KUKA KRL program: nplacestr5RS2.src, nplacestr5RS2.dat

--- nplacestr5RS2.src ---
&ACCESS RVP
&REL 1
&PARAM TEMPLATE = C:\KRC\Roboter\Template\ExpertVorgabe
&PARAM EDITMASK = *
DEF nplacestr5RS2( )
;FOLD INI
  ;FOLD BASISTECH INI
    GLOBAL INTERRUPT DECL 3 WHEN $STOPMESS==TRUE DO IR_STOPM ( )
    INTERRUPT ON 3
    BAS (#INITMOV,0 )
  ;ENDFOLD (BASISTECH INI)
  ;FOLD USER INI
    ;Make your modifications here

  ;ENDFOLD (USER INI)
;ENDFOLD (INI)




SWITCH NumCuring

;*******************************************************
CASE 90501
;*******************************************************
;*** Utilizar para hacer touchup en ptp a continuacion ***;
; 1  Ejecutar Axis_Rob_Move
; 2  Hacer TouchUp en ptp
; 3  Eliminar Axis_Rob_Move y comentarios

Axis_Rob_Move(1.69,-82.8,66.93,14.32,12.14,193,70,50)

;FOLD PTP pWB90501RS2 Vel=100 % PDAT_MESA Tool[10]:AMF1_G1000 Base[9]:BWB2S2;%{PE}%R 5.5.32,%MKUKATPBASIS,%CMOVE,%VPTP,%P 1:PTP, 2:pWB90501RS2, 3:, 5:100, 7:PDAT_MESA
$BWDSTART=FALSE
PDAT_ACT=PPDAT_MESA
FDAT_ACT=FpWB90501RS2
BAS(#PTP_PARAMS,100)
PTP XpWB90501RS2
;ENDFOLD
;*********************************************************;

;***Axis_Rob_Move de ayuda para aproximarse a dejada ***;
; Borrar tras touchup en LIN de dejada
Axis_Rob_Move(-90.22,-57.13,49.23,-5.44,97.37,193.9,20,50)
;*******************************************************;

PTP_OFFS(XP90501RS2, FP90501RS2, 0, -450, 30, 0, 0, 0, #TOOL, 20, 50, 0.0)

Cicle_Grp_M1000 (Inic_Pla_Right)

;***borrar***;
cyltopos(prg_200)
halt
;************;

LIN_OFFS(XP90501RS2, FP90501RS2, 0, 0, 30, 0, 0, 0, #TOOL, 0.1, 50, 0.0)
LIN_OFFS(XP90501RS2, FP90501RS2, 0, 0, 15, 0, 0, 0, #TOOL, 0.1, 50, 0.0)

Cntr_Grp_M1000 (C05C06,RH)

;FOLD LIN P90501RS2 Vel=0.1 m/s LV020Z0 Tool[10]:AMF1_G1000 Base[9]:BWB2S2;%{PE}%R 5.5.32,%MKUKATPBASIS,%CMOVE,%VLIN,%P 1:LIN, 2:P90501RS2, 3:, 5:0.1, 7:V020Z0
$BWDSTART=FALSE
LDAT_ACT=LV020Z0
FDAT_ACT=FP90501RS2
BAS(#CP_PARAMS,0.1)
LIN XP90501RS2
;ENDFOLD

Cntr_Grp_M1000 (AMF09,RLS)
Cyltopos (PRG_51)
Cntr_Grp_M1000 (C07C08,RH)
Cyltopos (PRG_61)
Cntr_Grp_M1000 (AMF10,RLS)
Cntr_Grp_M1000 (C05C06,FREE)
Cntr_Grp_M1000 (C07C08,FREE)
Cyltopos(PRG_88)
LIN_REL{Z -20}#TOOL
Cyltopos (PRG_105)
LIN_REL{Z -30}#TOOL
Cyltopos (PRG_200)

;*** MOVIMIENTOS DE OFFSETS ***;

LIN_OFFS(XP90501RS2, FP90501RS2, 0, 0, -50, 0, 0, 0, #TOOL, 0.3, 50, 0.0)
LIN_OFFS(XP90501RS2, FP90501RS2, 0, -450, -50, 0, 0, 0, #TOOL, 0.3, 50, 0.0)


;******* MEDICION LASER *******;

LIN_OFFS(XPLAS90501RS2_1, FPLAS90501RS2_1, 0, -200, 0, 0, 0, 0, #TOOL, 0.3, 50, 0.0)

cyltopos (prg_61)

;FOLD LIN PLAS90501RS2_1 Vel=0.3 m/s LV020Z0 Tool[10]:AMF1_G1000 Base[9]:BWB2S2;%{PE}%R 5.5.32,%MKUKATPBASIS,%CMOVE,%VLIN,%P 1:LIN, 2:PLAS90501RS2_1, 3:, 5:0.3, 7:V020Z0
$BWDSTART=FALSE
LDAT_ACT=LV020Z0
FDAT_ACT=FPLAS90501RS2_1
BAS(#CP_PARAMS,0.3)
LIN XPLAS90501RS2_1
;ENDFOLD

;Movimimiento de busqueda con laser
;Search( , )

;FOLD LIN PLAS90501RS2_2 Vel=0.3 m/s LV020Z0 Tool[10]:AMF1_G1000 Base[9]:BWB2S2;%{PE}%R 5.5.32,%MKUKATPBASIS,%CMOVE,%VLIN,%P 1:LIN, 2:PLAS90501RS2_2, 3:, 5:0.3, 7:V020Z0
$BWDSTART=FALSE
LDAT_ACT=LV020Z0
FDAT_ACT=FPLAS90501RS2_2
BAS(#CP_PARAMS,0.3)
LIN XPLAS90501RS2_2
;ENDFOLD


;Movimimiento de busqueda con laser
;Search( , )

LIN_OFFS(XPLAS90501RS2_1, FPLAS90501RS2_1, 0, -200, 0, 0, 0, 0, #TOOL, 0.3, 50, 0.0)

;******************************;

;FOLD PTP pWB90501RS2 Vel=100 % PDAT_MESA Tool[10]:AMF1_G1000 Base[9]:BWB2S2;%{PE}%R 5.5.32,%MKUKATPBASIS,%CMOVE,%VPTP,%P 1:PTP, 2:pWB90501RS2, 3:, 5:100, 7:PDAT_MESA
$BWDSTART=FALSE
PDAT_ACT=PPDAT_MESA
FDAT_ACT=FpWB90501RS2
BAS(#PTP_PARAMS,100)
PTP XpWB90501RS2
;ENDFOLD

;*******************************************************
CASE 90503
;*******************************************************
;*** Utilizar para hacer touchup en ptp a continuacion ***;
; 1  Ejecutar Axis_Rob_Move
; 2  Hacer TouchUp en ptp
; 3  Eliminar Axis_Rob_Move y comentarios

Axis_Rob_Move(1.69,-82.8,66.93,14.32,12.14,193,70,50)

;FOLD PTP pWB90503RS2 Vel=100 % PDAT_MESA Tool[10]:AMF1_G1000 Base[9]:BWB2S2;%{PE}%R 5.5.32,%MKUKATPBASIS,%CMOVE,%VPTP,%P 1:PTP, 2:pWB90503RS2, 3:, 5:100, 7:PDAT_MESA
$BWDSTART=FALSE
PDAT_ACT=PPDAT_MESA
FDAT_ACT=FpWB90503RS2
BAS(#PTP_PARAMS,100)
PTP XpWB90503RS2
;ENDFOLD
;*********************************************************;

;***Axis_Rob_Move de ayuda para aproximarse a dejada ***;
; Borrar tras touchup en LIN de dejada
Axis_Rob_Move(-90.22,-57.13,49.23,-5.44,97.37,193.9,20,50)
;*******************************************************;

PTP_OFFS(XP90503RS2, FP90503RS2, 0, -450, 30, 0, 0, 0, #TOOL, 20, 50, 0.0)

Cicle_Grp_M1000 (Inic_Pla_Right)

;***borrar***;
cyltopos(prg_200)
halt
;************;

LIN_OFFS(XP90503RS2, FP90503RS2, 0, 0, 30, 0, 0, 0, #TOOL, 0.1, 50, 0.0)
LIN_OFFS(XP90503RS2, FP90503RS2, 0, 0, 15, 0, 0, 0, #TOOL, 0.1, 50, 0.0)

Cntr_Grp_M1000 (C05C06,RH)

;FOLD LIN P90503RS2 Vel=0.1 m/s LV020Z0 Tool[10]:AMF1_G1000 Base[9]:BWB2S2;%{PE}%R 5.5.32,%MKUKATPBASIS,%CMOVE,%VLIN,%P 1:LIN, 2:P90503RS2, 3:, 5:0.1, 7:V020Z0
$BWDSTART=FALSE
LDAT_ACT=LV020Z0
FDAT_ACT=FP90503RS2
BAS(#CP_PARAMS,0.1)
LIN XP90503RS2
;ENDFOLD

Cntr_Grp_M1000 (AMF09,RLS)
Cyltopos (PRG_51)
Cntr_Grp_M1000 (C07C08,RH)
Cyltopos (PRG_61)
Cntr_Grp_M1000 (AMF10,RLS)
Cntr_Grp_M1000 (C05C06,FREE)
Cntr_Grp_M1000 (C07C08,FREE)
Cyltopos(PRG_88)
LIN_REL{Z -20}#TOOL
Cyltopos (PRG_105)
LIN_REL{Z -30}#TOOL
Cyltopos (PRG_200)

;*** MOVIMIENTOS DE OFFSETS ***;

LIN_OFFS(XP90503RS2, FP90503RS2, 0, 0, -50, 0, 0, 0, #TOOL, 0.3, 50, 0.0)
LIN_OFFS(XP90503RS2, FP90503RS2, 0, -450, -50, 0, 0, 0, #TOOL, 0.3, 50, 0.0)


;******* MEDICION LASER *******;

LIN_OFFS(XPLAS90503RS2_1, FPLAS90503RS2_1, 0, -200, 0, 0, 0, 0, #TOOL, 0.3, 50, 0.0)

cyltopos (prg_61)

;FOLD LIN PLAS90503RS2_1 Vel=0.3 m/s LV020Z0 Tool[10]:AMF1_G1000 Base[9]:BWB2S2;%{PE}%R 5.5.32,%MKUKATPBASIS,%CMOVE,%VLIN,%P 1:LIN, 2:PLAS90503RS2_1, 3:, 5:0.3, 7:V020Z0
$BWDSTART=FALSE
LDAT_ACT=LV020Z0
FDAT_ACT=FPLAS90503RS2_1
BAS(#CP_PARAMS,0.3)
LIN XPLAS90503RS2_1
;ENDFOLD

;Movimimiento de busqueda con laser
;Search( , )

;FOLD LIN PLAS90503RS2_2 Vel=0.3 m/s LV020Z0 Tool[10]:AMF1_G1000 Base[9]:BWB2S2;%{PE}%R 5.5.32,%MKUKATPBASIS,%CMOVE,%VLIN,%P 1:LIN, 2:PLAS90503RS2_2, 3:, 5:0.3, 7:V020Z0
$BWDSTART=FALSE
LDAT_ACT=LV020Z0
FDAT_ACT=FPLAS90503RS2_2
BAS(#CP_PARAMS,0.3)
LIN XPLAS90503RS2_2
;ENDFOLD


;Movimimiento de busqueda con laser
;Search( , )

LIN_OFFS(XPLAS90503RS2_1, FPLAS90503RS2_1, 0, -200, 0, 0, 0, 0, #TOOL, 0.3, 50, 0.0)

;******************************;

;FOLD PTP pWB90503RS2 Vel=100 % PDAT_MESA Tool[10]:AMF1_G1000 Base[9]:BWB2S2;%{PE}%R 5.5.32,%MKUKATPBASIS,%CMOVE,%VPTP,%P 1:PTP, 2:pWB90503RS2, 3:, 5:100, 7:PDAT_MESA
$BWDSTART=FALSE
PDAT_ACT=PPDAT_MESA
FDAT_ACT=FpWB90503RS2
BAS(#PTP_PARAMS,100)
PTP XpWB90503RS2
;ENDFOLD

;*******************************************************
CASE 90505
;*******************************************************
;*** Utilizar para hacer touchup en ptp a continuacion ***;
; 1  Ejecutar Axis_Rob_Move
; 2  Hacer TouchUp en ptp
; 3  Eliminar Axis_Rob_Move y comentarios

Axis_Rob_Move(1.69,-82.8,66.93,14.32,12.14,193,70,50)

;FOLD PTP pWB90505RS2 Vel=100 % PDAT_MESA Tool[10]:AMF1_G1000 Base[9]:BWB2S2;%{PE}%R 5.5.32,%MKUKATPBASIS,%CMOVE,%VPTP,%P 1:PTP, 2:pWB90505RS2, 3:, 5:100, 7:PDAT_MESA
$BWDSTART=FALSE
PDAT_ACT=PPDAT_MESA
FDAT_ACT=FpWB90505RS2
BAS(#PTP_PARAMS,100)
PTP XpWB90505RS2
;ENDFOLD
;*********************************************************;

;***Axis_Rob_Move de ayuda para aproximarse a dejada ***;
; Borrar tras touchup en LIN de dejada
Axis_Rob_Move(-90.22,-57.13,49.23,-5.44,97.37,193.9,20,50)
;*******************************************************;

PTP_OFFS(XP90505RS2, FP90505RS2, 0, -450, 30, 0, 0, 0, #TOOL, 20, 50, 0.0)

Cicle_Grp_M1000 (Inic_Pla_Right)

;***borrar***;
cyltopos(prg_200)
halt
;************;

LIN_OFFS(XP90505RS2, FP90505RS2, 0, 0, 30, 0, 0, 0, #TOOL, 0.1, 50, 0.0)
LIN_OFFS(XP90505RS2, FP90505RS2, 0, 0, 15, 0, 0, 0, #TOOL, 0.1, 50, 0.0)

Cntr_Grp_M1000 (C05C06,RH)

;FOLD LIN P90505RS2 Vel=0.1 m/s LV020Z0 Tool[10]:AMF1_G1000 Base[9]:BWB2S2;%{PE}%R 5.5.32,%MKUKATPBASIS,%CMOVE,%VLIN,%P 1:LIN, 2:P90505RS2, 3:, 5:0.1, 7:V020Z0
$BWDSTART=FALSE
LDAT_ACT=LV020Z0
FDAT_ACT=FP90505RS2
BAS(#CP_PARAMS,0.1)
LIN XP90505RS2
;ENDFOLD

Cntr_Grp_M1000 (AMF09,RLS)
Cyltopos (PRG_51)
Cntr_Grp_M1000 (C07C08,RH)
Cyltopos (PRG_61)
Cntr_Grp_M1000 (AMF10,RLS)
Cntr_Grp_M1000 (C05C06,FREE)
Cntr_Grp_M1000 (C07C08,FREE)
Cyltopos(PRG_88)
LIN_REL{Z -20}#TOOL
Cyltopos (PRG_105)
LIN_REL{Z -30}#TOOL
Cyltopos (PRG_200)

;*** MOVIMIENTOS DE OFFSETS ***;

LIN_OFFS(XP90505RS2, FP90505RS2, 0, 0, -50, 0, 0, 0, #TOOL, 0.3, 50, 0.0)
LIN_OFFS(XP90505RS2, FP90505RS2, 0, -450, -50, 0, 0, 0, #TOOL, 0.3, 50, 0.0)


;******* MEDICION LASER *******;

LIN_OFFS(XPLAS90505RS2_1, FPLAS90505RS2_1, 0, -200, 0, 0, 0, 0, #TOOL, 0.3, 50, 0.0)

cyltopos (prg_61)

;FOLD LIN PLAS90505RS2_1 Vel=0.3 m/s LV020Z0 Tool[10]:AMF1_G1000 Base[9]:BWB2S2;%{PE}%R 5.5.32,%MKUKATPBASIS,%CMOVE,%VLIN,%P 1:LIN, 2:PLAS90505RS2_1, 3:, 5:0.3, 7:V020Z0
$BWDSTART=FALSE
LDAT_ACT=LV020Z0
FDAT_ACT=FPLAS90505RS2_1
BAS(#CP_PARAMS,0.3)
LIN XPLAS90505RS2_1
;ENDFOLD

;Movimimiento de busqueda con laser
;Search( , )

;FOLD LIN PLAS90505RS2_2 Vel=0.3 m/s LV020Z0 Tool[10]:AMF1_G1000 Base[9]:BWB2S2;%{PE}%R 5.5.32,%MKUKATPBASIS,%CMOVE,%VLIN,%P 1:LIN, 2:PLAS90505RS2_2, 3:, 5:0.3, 7:V020Z0
$BWDSTART=FALSE
LDAT_ACT=LV020Z0
FDAT_ACT=FPLAS90505RS2_2
BAS(#CP_PARAMS,0.3)
LIN XPLAS90505RS2_2
;ENDFOLD


;Movimimiento de busqueda con laser
;Search( , )

LIN_OFFS(XPLAS90505RS2_1, FPLAS90505RS2_1, 0, -200, 0, 0, 0, 0, #TOOL, 0.3, 50, 0.0)

;******************************;

;FOLD PTP pWB90505RS2 Vel=100 % PDAT_MESA Tool[10]:AMF1_G1000 Base[9]:BWB2S2;%{PE}%R 5.5.32,%MKUKATPBASIS,%CMOVE,%VPTP,%P 1:PTP, 2:pWB90505RS2, 3:, 5:100, 7:PDAT_MESA
$BWDSTART=FALSE
PDAT_ACT=PPDAT_MESA
FDAT_ACT=FpWB90505RS2
BAS(#PTP_PARAMS,100)
PTP XpWB90505RS2
;ENDFOLD

;*******************************************************
CASE 90507
;*******************************************************
;*** Utilizar para hacer touchup en ptp a continuacion ***;
; 1  Ejecutar Axis_Rob_Move
; 2  Hacer TouchUp en ptp
; 3  Eliminar Axis_Rob_Move y comentarios

Axis_Rob_Move(1.69,-82.8,66.93,14.32,12.14,193,70,50)

;FOLD PTP pWB90507RS2 Vel=100 % PDAT_MESA Tool[10]:AMF1_G1000 Base[9]:BWB2S2;%{PE}%R 5.5.32,%MKUKATPBASIS,%CMOVE,%VPTP,%P 1:PTP, 2:pWB90507RS2, 3:, 5:100, 7:PDAT_MESA
$BWDSTART=FALSE
PDAT_ACT=PPDAT_MESA
FDAT_ACT=FpWB90507RS2
BAS(#PTP_PARAMS,100)
PTP XpWB90507RS2
;ENDFOLD
;*********************************************************;

;***Axis_Rob_Move de ayuda para aproximarse a dejada ***;
; Borrar tras touchup en LIN de dejada
Axis_Rob_Move(-90.22,-57.13,49.23,-5.44,97.37,193.9,20,50)
;*******************************************************;

PTP_OFFS(XP90507RS2, FP90507RS2, 0, -450, 30, 0, 0, 0, #TOOL, 20, 50, 0.0)

Cicle_Grp_M1000 (Inic_Pla_Right)

;***borrar***;
cyltopos(prg_200)
halt
;************;

LIN_OFFS(XP90507RS2, FP90507RS2, 0, 0, 30, 0, 0, 0, #TOOL, 0.1, 50, 0.0)
LIN_OFFS(XP90507RS2, FP90507RS2, 0, 0, 15, 0, 0, 0, #TOOL, 0.1, 50, 0.0)

Cntr_Grp_M1000 (C05C06,RH)

;FOLD LIN P90507RS2 Vel=0.1 m/s LV020Z0 Tool[10]:AMF1_G1000 Base[9]:BWB2S2;%{PE}%R 5.5.32,%MKUKATPBASIS,%CMOVE,%VLIN,%P 1:LIN, 2:P90507RS2, 3:, 5:0.1, 7:V020Z0
$BWDSTART=FALSE
LDAT_ACT=LV020Z0
FDAT_ACT=FP90507RS2
BAS(#CP_PARAMS,0.1)
LIN XP90507RS2
;ENDFOLD

Cntr_Grp_M1000 (AMF09,RLS)
Cyltopos (PRG_51)
Cntr_Grp_M1000 (C07C08,RH)
Cyltopos (PRG_61)
Cntr_Grp_M1000 (AMF10,RLS)
Cntr_Grp_M1000 (C05C06,FREE)
Cntr_Grp_M1000 (C07C08,FREE)
Cyltopos(PRG_88)
LIN_REL{Z -20}#TOOL
Cyltopos (PRG_105)
LIN_REL{Z -30}#TOOL
Cyltopos (PRG_200)

;*** MOVIMIENTOS DE OFFSETS ***;

LIN_OFFS(XP90507RS2, FP90507RS2, 0, 0, -50, 0, 0, 0, #TOOL, 0.3, 50, 0.0)
LIN_OFFS(XP90507RS2, FP90507RS2, 0, -450, -50, 0, 0, 0, #TOOL, 0.3, 50, 0.0)


;******* MEDICION LASER *******;

LIN_OFFS(XPLAS90507RS2_1, FPLAS90507RS2_1, 0, -200, 0, 0, 0, 0, #TOOL, 0.3, 50, 0.0)

cyltopos (prg_61)

;FOLD LIN PLAS90507RS2_1 Vel=0.3 m/s LV020Z0 Tool[10]:AMF1_G1000 Base[9]:BWB2S2;%{PE}%R 5.5.32,%MKUKATPBASIS,%CMOVE,%VLIN,%P 1:LIN, 2:PLAS90507RS2_1, 3:, 5:0.3, 7:V020Z0
$BWDSTART=FALSE
LDAT_ACT=LV020Z0
FDAT_ACT=FPLAS90507RS2_1
BAS(#CP_PARAMS,0.3)
LIN XPLAS90507RS2_1
;ENDFOLD

;Movimimiento de busqueda con laser
;Search( , )

;FOLD LIN PLAS90507RS2_2 Vel=0.3 m/s LV020Z0 Tool[10]:AMF1_G1000 Base[9]:BWB2S2;%{PE}%R 5.5.32,%MKUKATPBASIS,%CMOVE,%VLIN,%P 1:LIN, 2:PLAS90507RS2_2, 3:, 5:0.3, 7:V020Z0
$BWDSTART=FALSE
LDAT_ACT=LV020Z0
FDAT_ACT=FPLAS90507RS2_2
BAS(#CP_PARAMS,0.3)
LIN XPLAS90507RS2_2
;ENDFOLD


;Movimimiento de busqueda con laser
;Search( , )

LIN_OFFS(XPLAS90507RS2_1, FPLAS90507RS2_1, 0, -200, 0, 0, 0, 0, #TOOL, 0.3, 50, 0.0)

;******************************;

;FOLD PTP pWB90507RS2 Vel=100 % PDAT_MESA Tool[10]:AMF1_G1000 Base[9]:BWB2S2;%{PE}%R 5.5.32,%MKUKATPBASIS,%CMOVE,%VPTP,%P 1:PTP, 2:pWB90507RS2, 3:, 5:100, 7:PDAT_MESA
$BWDSTART=FALSE
PDAT_ACT=PPDAT_MESA
FDAT_ACT=FpWB90507RS2
BAS(#PTP_PARAMS,100)
PTP XpWB90507RS2
;ENDFOLD

;*******************************************************
CASE 90509
;*******************************************************
;*** Utilizar para hacer touchup en ptp a continuacion ***;
; 1  Ejecutar Axis_Rob_Move
; 2  Hacer TouchUp en ptp
; 3  Eliminar Axis_Rob_Move y comentarios

Axis_Rob_Move(1.69,-82.8,66.93,14.32,12.14,193,70,50)

;FOLD PTP pWB90509RS2 Vel=100 % PDAT_MESA Tool[10]:AMF1_G1000 Base[9]:BWB2S2;%{PE}%R 5.5.32,%MKUKATPBASIS,%CMOVE,%VPTP,%P 1:PTP, 2:pWB90509RS2, 3:, 5:100, 7:PDAT_MESA
$BWDSTART=FALSE
PDAT_ACT=PPDAT_MESA
FDAT_ACT=FpWB90509RS2
BAS(#PTP_PARAMS,100)
PTP XpWB90509RS2
;ENDFOLD
;*********************************************************;

;***Axis_Rob_Move de ayuda para aproximarse a dejada ***;
; Borrar tras touchup en LIN de dejada
Axis_Rob_Move(-90.22,-57.13,49.23,-5.44,97.37,193.9,20,50)
;*******************************************************;

PTP_OFFS(XP90509RS2, FP90509RS2, 0, -450, 30, 0, 0, 0, #TOOL, 20, 50, 0.0)

Cicle_Grp_M1000 (Inic_Pla_Right)

;***borrar***;
cyltopos(prg_200)
halt
;************;

LIN_OFFS(XP90509RS2, FP90509RS2, 0, 0, 30, 0, 0, 0, #TOOL, 0.1, 50, 0.0)
LIN_OFFS(XP90509RS2, FP90509RS2, 0, 0, 15, 0, 0, 0, #TOOL, 0.1, 50, 0.0)

Cntr_Grp_M1000 (C05C06,RH)

;FOLD LIN P90509RS2 Vel=0.1 m/s LV020Z0 Tool[10]:AMF1_G1000 Base[9]:BWB2S2;%{PE}%R 5.5.32,%MKUKATPBASIS,%CMOVE,%VLIN,%P 1:LIN, 2:P90509RS2, 3:, 5:0.1, 7:V020Z0
$BWDSTART=FALSE
LDAT_ACT=LV020Z0
FDAT_ACT=FP90509RS2
BAS(#CP_PARAMS,0.1)
LIN XP90509RS2
;ENDFOLD

Cntr_Grp_M1000 (AMF09,RLS)
Cyltopos (PRG_51)
Cntr_Grp_M1000 (C07C08,RH)
Cyltopos (PRG_61)
Cntr_Grp_M1000 (AMF10,RLS)
Cntr_Grp_M1000 (C05C06,FREE)
Cntr_Grp_M1000 (C07C08,FREE)
Cyltopos(PRG_88)
LIN_REL{Z -20}#TOOL
Cyltopos (PRG_105)
LIN_REL{Z -30}#TOOL
Cyltopos (PRG_200)

;*** MOVIMIENTOS DE OFFSETS ***;

LIN_OFFS(XP90509RS2, FP90509RS2, 0, 0, -50, 0, 0, 0, #TOOL, 0.3, 50, 0.0)
LIN_OFFS(XP90509RS2, FP90509RS2, 0, -450, -50, 0, 0, 0, #TOOL, 0.3, 50, 0.0)


;******* MEDICION LASER *******;

LIN_OFFS(XPLAS90509RS2_1, FPLAS90509RS2_1, 0, -200, 0, 0, 0, 0, #TOOL, 0.3, 50, 0.0)

cyltopos (prg_61)

;FOLD LIN PLAS90509RS2_1 Vel=0.3 m/s LV020Z0 Tool[10]:AMF1_G1000 Base[9]:BWB2S2;%{PE}%R 5.5.32,%MKUKATPBASIS,%CMOVE,%VLIN,%P 1:LIN, 2:PLAS90509RS2_1, 3:, 5:0.3, 7:V020Z0
$BWDSTART=FALSE
LDAT_ACT=LV020Z0
FDAT_ACT=FPLAS90509RS2_1
BAS(#CP_PARAMS,0.3)
LIN XPLAS90509RS2_1
;ENDFOLD

;Movimimiento de busqueda con laser
;Search( , )

;FOLD LIN PLAS90509RS2_2 Vel=0.3 m/s LV020Z0 Tool[10]:AMF1_G1000 Base[9]:BWB2S2;%{PE}%R 5.5.32,%MKUKATPBASIS,%CMOVE,%VLIN,%P 1:LIN, 2:PLAS90509RS2_2, 3:, 5:0.3, 7:V020Z0
$BWDSTART=FALSE
LDAT_ACT=LV020Z0
FDAT_ACT=FPLAS90509RS2_2
BAS(#CP_PARAMS,0.3)
LIN XPLAS90509RS2_2
;ENDFOLD


;Movimimiento de busqueda con laser
;Search( , )

LIN_OFFS(XPLAS90509RS2_1, FPLAS90509RS2_1, 0, -200, 0, 0, 0, 0, #TOOL, 0.3, 50, 0.0)

;******************************;

;FOLD PTP pWB90509RS2 Vel=100 % PDAT_MESA Tool[10]:AMF1_G1000 Base[9]:BWB2S2;%{PE}%R 5.5.32,%MKUKATPBASIS,%CMOVE,%VPTP,%P 1:PTP, 2:pWB90509RS2, 3:, 5:100, 7:PDAT_MESA
$BWDSTART=FALSE
PDAT_ACT=PPDAT_MESA
FDAT_ACT=FpWB90509RS2
BAS(#PTP_PARAMS,100)
PTP XpWB90509RS2
;ENDFOLD

;*******************************************************
CASE 90511
;*******************************************************
;*** Utilizar para hacer touchup en ptp a continuacion ***;
; 1  Ejecutar Axis_Rob_Move
; 2  Hacer TouchUp en ptp
; 3  Eliminar Axis_Rob_Move y comentarios

Axis_Rob_Move(1.69,-82.8,66.93,14.32,12.14,193,70,50)

;FOLD PTP pWB90511RS2 Vel=100 % PDAT_MESA Tool[10]:AMF1_G1000 Base[9]:BWB2S2;%{PE}%R 5.5.32,%MKUKATPBASIS,%CMOVE,%VPTP,%P 1:PTP, 2:pWB90511RS2, 3:, 5:100, 7:PDAT_MESA
$BWDSTART=FALSE
PDAT_ACT=PPDAT_MESA
FDAT_ACT=FpWB90511RS2
BAS(#PTP_PARAMS,100)
PTP XpWB90511RS2
;ENDFOLD
;*********************************************************;

;***Axis_Rob_Move de ayuda para aproximarse a dejada ***;
; Borrar tras touchup en LIN de dejada
Axis_Rob_Move(-90.22,-57.13,49.23,-5.44,97.37,193.9,20,50)
;*******************************************************;

PTP_OFFS(XP90511RS2, FP90511RS2, 0, -450, 30, 0, 0, 0, #TOOL, 20, 50, 0.0)

Cicle_Grp_M1000 (Inic_Pla_Right)

;***borrar***;
cyltopos(prg_200)
halt
;************;

LIN_OFFS(XP90511RS2, FP90511RS2, 0, 0, 30, 0, 0, 0, #TOOL, 0.1, 50, 0.0)
LIN_OFFS(XP90511RS2, FP90511RS2, 0, 0, 15, 0, 0, 0, #TOOL, 0.1, 50, 0.0)

Cntr_Grp_M1000 (C05C06,RH)

;FOLD LIN P90511RS2 Vel=0.1 m/s LV020Z0 Tool[10]:AMF1_G1000 Base[9]:BWB2S2;%{PE}%R 5.5.32,%MKUKATPBASIS,%CMOVE,%VLIN,%P 1:LIN, 2:P90511RS2, 3:, 5:0.1, 7:V020Z0
$BWDSTART=FALSE
LDAT_ACT=LV020Z0
FDAT_ACT=FP90511RS2
BAS(#CP_PARAMS,0.1)
LIN XP90511RS2
;ENDFOLD

Cntr_Grp_M1000 (AMF09,RLS)
Cyltopos (PRG_51)
Cntr_Grp_M1000 (C07C08,RH)
Cyltopos (PRG_61)
Cntr_Grp_M1000 (AMF10,RLS)
Cntr_Grp_M1000 (C05C06,FREE)
Cntr_Grp_M1000 (C07C08,FREE)
Cyltopos(PRG_88)
LIN_REL{Z -20}#TOOL
Cyltopos (PRG_105)
LIN_REL{Z -30}#TOOL
Cyltopos (PRG_200)

;*** MOVIMIENTOS DE OFFSETS ***;

LIN_OFFS(XP90511RS2, FP90511RS2, 0, 0, -50, 0, 0, 0, #TOOL, 0.3, 50, 0.0)
LIN_OFFS(XP90511RS2, FP90511RS2, 0, -450, -50, 0, 0, 0, #TOOL, 0.3, 50, 0.0)


;******* MEDICION LASER *******;

LIN_OFFS(XPLAS90511RS2_1, FPLAS90511RS2_1, 0, -200, 0, 0, 0, 0, #TOOL, 0.3, 50, 0.0)

cyltopos (prg_61)

;FOLD LIN PLAS90511RS2_1 Vel=0.3 m/s LV020Z0 Tool[10]:AMF1_G1000 Base[9]:BWB2S2;%{PE}%R 5.5.32,%MKUKATPBASIS,%CMOVE,%VLIN,%P 1:LIN, 2:PLAS90511RS2_1, 3:, 5:0.3, 7:V020Z0
$BWDSTART=FALSE
LDAT_ACT=LV020Z0
FDAT_ACT=FPLAS90511RS2_1
BAS(#CP_PARAMS,0.3)
LIN XPLAS90511RS2_1
;ENDFOLD

;Movimimiento de busqueda con laser
;Search( , )

;FOLD LIN PLAS90511RS2_2 Vel=0.3 m/s LV020Z0 Tool[10]:AMF1_G1000 Base[9]:BWB2S2;%{PE}%R 5.5.32,%MKUKATPBASIS,%CMOVE,%VLIN,%P 1:LIN, 2:PLAS90511RS2_2, 3:, 5:0.3, 7:V020Z0
$BWDSTART=FALSE
LDAT_ACT=LV020Z0
FDAT_ACT=FPLAS90511RS2_2
BAS(#CP_PARAMS,0.3)
LIN XPLAS90511RS2_2
;ENDFOLD


;Movimimiento de busqueda con laser
;Search( , )

LIN_OFFS(XPLAS90511RS2_1, FPLAS90511RS2_1, 0, -200, 0, 0, 0, 0, #TOOL, 0.3, 50, 0.0)

;******************************;

;FOLD PTP pWB90511RS2 Vel=100 % PDAT_MESA Tool[10]:AMF1_G1000 Base[9]:BWB2S2;%{PE}%R 5.5.32,%MKUKATPBASIS,%CMOVE,%VPTP,%P 1:PTP, 2:pWB90511RS2, 3:, 5:100, 7:PDAT_MESA
$BWDSTART=FALSE
PDAT_ACT=PPDAT_MESA
FDAT_ACT=FpWB90511RS2
BAS(#PTP_PARAMS,100)
PTP XpWB90511RS2
;ENDFOLD

;*******************************************************
CASE 90513
;*******************************************************
;*** Utilizar para hacer touchup en ptp a continuacion ***;
; 1  Ejecutar Axis_Rob_Move
; 2  Hacer TouchUp en ptp
; 3  Eliminar Axis_Rob_Move y comentarios

Axis_Rob_Move(1.69,-82.8,66.93,14.32,12.14,193,70,50)

;FOLD PTP pWB90513RS2 Vel=100 % PDAT_MESA Tool[10]:AMF1_G1000 Base[9]:BWB2S2;%{PE}%R 5.5.32,%MKUKATPBASIS,%CMOVE,%VPTP,%P 1:PTP, 2:pWB90513RS2, 3:, 5:100, 7:PDAT_MESA
$BWDSTART=FALSE
PDAT_ACT=PPDAT_MESA
FDAT_ACT=FpWB90513RS2
BAS(#PTP_PARAMS,100)
PTP XpWB90513RS2
;ENDFOLD
;*********************************************************;

;***Axis_Rob_Move de ayuda para aproximarse a dejada ***;
; Borrar tras touchup en LIN de dejada
Axis_Rob_Move(-90.22,-57.13,49.23,-5.44,97.37,193.9,20,50)
;*******************************************************;

PTP_OFFS(XP90513RS2, FP90513RS2, 0, -450, 30, 0, 0, 0, #TOOL, 20, 50, 0.0)

Cicle_Grp_M1000 (Inic_Pla_Right)

;***borrar***;
cyltopos(prg_200)
halt
;************;

LIN_OFFS(XP90513RS2, FP90513RS2, 0, 0, 30, 0, 0, 0, #TOOL, 0.1, 50, 0.0)
LIN_OFFS(XP90513RS2, FP90513RS2, 0, 0, 15, 0, 0, 0, #TOOL, 0.1, 50, 0.0)

Cntr_Grp_M1000 (C05C06,RH)

;FOLD LIN P90513RS2 Vel=0.1 m/s LV020Z0 Tool[10]:AMF1_G1000 Base[9]:BWB2S2;%{PE}%R 5.5.32,%MKUKATPBASIS,%CMOVE,%VLIN,%P 1:LIN, 2:P90513RS2, 3:, 5:0.1, 7:V020Z0
$BWDSTART=FALSE
LDAT_ACT=LV020Z0
FDAT_ACT=FP90513RS2
BAS(#CP_PARAMS,0.1)
LIN XP90513RS2
;ENDFOLD

Cntr_Grp_M1000 (AMF09,RLS)
Cyltopos (PRG_51)
Cntr_Grp_M1000 (C07C08,RH)
Cyltopos (PRG_61)
Cntr_Grp_M1000 (AMF10,RLS)
Cntr_Grp_M1000 (C05C06,FREE)
Cntr_Grp_M1000 (C07C08,FREE)
Cyltopos(PRG_88)
LIN_REL{Z -20}#TOOL
Cyltopos (PRG_105)
LIN_REL{Z -30}#TOOL
Cyltopos (PRG_200)

;*** MOVIMIENTOS DE OFFSETS ***;

LIN_OFFS(XP90513RS2, FP90513RS2, 0, 0, -50, 0, 0, 0, #TOOL, 0.3, 50, 0.0)
LIN_OFFS(XP90513RS2, FP90513RS2, 0, -450, -50, 0, 0, 0, #TOOL, 0.3, 50, 0.0)


;******* MEDICION LASER *******;

LIN_OFFS(XPLAS90513RS2_1, FPLAS90513RS2_1, 0, -200, 0, 0, 0, 0, #TOOL, 0.3, 50, 0.0)

cyltopos (prg_61)

;FOLD LIN PLAS90513RS2_1 Vel=0.3 m/s LV020Z0 Tool[10]:AMF1_G1000 Base[9]:BWB2S2;%{PE}%R 5.5.32,%MKUKATPBASIS,%CMOVE,%VLIN,%P 1:LIN, 2:PLAS90513RS2_1, 3:, 5:0.3, 7:V020Z0
$BWDSTART=FALSE
LDAT_ACT=LV020Z0
FDAT_ACT=FPLAS90513RS2_1
BAS(#CP_PARAMS,0.3)
LIN XPLAS90513RS2_1
;ENDFOLD

;Movimimiento de busqueda con laser
;Search( , )

;FOLD LIN PLAS90513RS2_2 Vel=0.3 m/s LV020Z0 Tool[10]:AMF1_G1000 Base[9]:BWB2S2;%{PE}%R 5.5.32,%MKUKATPBASIS,%CMOVE,%VLIN,%P 1:LIN, 2:PLAS90513RS2_2, 3:, 5:0.3, 7:V020Z0
$BWDSTART=FALSE
LDAT_ACT=LV020Z0
FDAT_ACT=FPLAS90513RS2_2
BAS(#CP_PARAMS,0.3)
LIN XPLAS90513RS2_2
;ENDFOLD


;Movimimiento de busqueda con laser
;Search( , )

LIN_OFFS(XPLAS90513RS2_1, FPLAS90513RS2_1, 0, -200, 0, 0, 0, 0, #TOOL, 0.3, 50, 0.0)

;******************************;

;FOLD PTP pWB90513RS2 Vel=100 % PDAT_MESA Tool[10]:AMF1_G1000 Base[9]:BWB2S2;%{PE}%R 5.5.32,%MKUKATPBASIS,%CMOVE,%VPTP,%P 1:PTP, 2:pWB90513RS2, 3:, 5:100, 7:PDAT_MESA
$BWDSTART=FALSE
PDAT_ACT=PPDAT_MESA
FDAT_ACT=FpWB90513RS2
BAS(#PTP_PARAMS,100)
PTP XpWB90513RS2
;ENDFOLD

;*******************************************************
CASE 90515
;*******************************************************
;*** Utilizar para hacer touchup en ptp a continuacion ***;
; 1  Ejecutar Axis_Rob_Move
; 2  Hacer TouchUp en ptp
; 3  Eliminar Axis_Rob_Move y comentarios

Axis_Rob_Move(1.69,-82.8,66.93,14.32,12.14,193,70,50)

;FOLD PTP pWB90515RS2 Vel=100 % PDAT_MESA Tool[10]:AMF1_G1000 Base[9]:BWB2S2;%{PE}%R 5.5.32,%MKUKATPBASIS,%CMOVE,%VPTP,%P 1:PTP, 2:pWB90515RS2, 3:, 5:100, 7:PDAT_MESA
$BWDSTART=FALSE
PDAT_ACT=PPDAT_MESA
FDAT_ACT=FpWB90515RS2
BAS(#PTP_PARAMS,100)
PTP XpWB90515RS2
;ENDFOLD
;*********************************************************;

;***Axis_Rob_Move de ayuda para aproximarse a dejada ***;
; Borrar tras touchup en LIN de dejada
Axis_Rob_Move(-90.22,-57.13,49.23,-5.44,97.37,193.9,20,50)
;*******************************************************;

PTP_OFFS(XP90515RS2, FP90515RS2, 0, -450, 30, 0, 0, 0, #TOOL, 20, 50, 0.0)

Cicle_Grp_M1000 (Inic_Pla_Right)

;***borrar***;
cyltopos(prg_200)
halt
;************;

LIN_OFFS(XP90515RS2, FP90515RS2, 0, 0, 30, 0, 0, 0, #TOOL, 0.1, 50, 0.0)
LIN_OFFS(XP90515RS2, FP90515RS2, 0, 0, 15, 0, 0, 0, #TOOL, 0.1, 50, 0.0)

Cntr_Grp_M1000 (C05C06,RH)

;FOLD LIN P90515RS2 Vel=0.1 m/s LV020Z0 Tool[10]:AMF1_G1000 Base[9]:BWB2S2;%{PE}%R 5.5.32,%MKUKATPBASIS,%CMOVE,%VLIN,%P 1:LIN, 2:P90515RS2, 3:, 5:0.1, 7:V020Z0
$BWDSTART=FALSE
LDAT_ACT=LV020Z0
FDAT_ACT=FP90515RS2
BAS(#CP_PARAMS,0.1)
LIN XP90515RS2
;ENDFOLD

Cntr_Grp_M1000 (AMF09,RLS)
Cyltopos (PRG_51)
Cntr_Grp_M1000 (C07C08,RH)
Cyltopos (PRG_61)
Cntr_Grp_M1000 (AMF10,RLS)
Cntr_Grp_M1000 (C05C06,FREE)
Cntr_Grp_M1000 (C07C08,FREE)
Cyltopos(PRG_88)
LIN_REL{Z -20}#TOOL
Cyltopos (PRG_105)
LIN_REL{Z -30}#TOOL
Cyltopos (PRG_200)

;*** MOVIMIENTOS DE OFFSETS ***;

LIN_OFFS(XP90515RS2, FP90515RS2, 0, 0, -50, 0, 0, 0, #TOOL, 0.3, 50, 0.0)
LIN_OFFS(XP90515RS2, FP90515RS2, 0, -450, -50, 0, 0, 0, #TOOL, 0.3, 50, 0.0)


;******* MEDICION LASER *******;

LIN_OFFS(XPLAS90515RS2_1, FPLAS90515RS2_1, 0, -200, 0, 0, 0, 0, #TOOL, 0.3, 50, 0.0)

cyltopos (prg_61)

;FOLD LIN PLAS90515RS2_1 Vel=0.3 m/s LV020Z0 Tool[10]:AMF1_G1000 Base[9]:BWB2S2;%{PE}%R 5.5.32,%MKUKATPBASIS,%CMOVE,%VLIN,%P 1:LIN, 2:PLAS90515RS2_1, 3:, 5:0.3, 7:V020Z0
$BWDSTART=FALSE
LDAT_ACT=LV020Z0
FDAT_ACT=FPLAS90515RS2_1
BAS(#CP_PARAMS,0.3)
LIN XPLAS90515RS2_1
;ENDFOLD

;Movimimiento de busqueda con laser
;Search( , )

;FOLD LIN PLAS90515RS2_2 Vel=0.3 m/s LV020Z0 Tool[10]:AMF1_G1000 Base[9]:BWB2S2;%{PE}%R 5.5.32,%MKUKATPBASIS,%CMOVE,%VLIN,%P 1:LIN, 2:PLAS90515RS2_2, 3:, 5:0.3, 7:V020Z0
$BWDSTART=FALSE
LDAT_ACT=LV020Z0
FDAT_ACT=FPLAS90515RS2_2
BAS(#CP_PARAMS,0.3)
LIN XPLAS90515RS2_2
;ENDFOLD


;Movimimiento de busqueda con laser
;Search( , )

LIN_OFFS(XPLAS90515RS2_1, FPLAS90515RS2_1, 0, -200, 0, 0, 0, 0, #TOOL, 0.3, 50, 0.0)

;******************************;

;FOLD PTP pWB90515RS2 Vel=100 % PDAT_MESA Tool[10]:AMF1_G1000 Base[9]:BWB2S2;%{PE}%R 5.5.32,%MKUKATPBASIS,%CMOVE,%VPTP,%P 1:PTP, 2:pWB90515RS2, 3:, 5:100, 7:PDAT_MESA
$BWDSTART=FALSE
PDAT_ACT=PPDAT_MESA
FDAT_ACT=FpWB90515RS2
BAS(#PTP_PARAMS,100)
PTP XpWB90515RS2
;ENDFOLD

;*******************************************************
CASE 90517
;*******************************************************
;*** Utilizar para hacer touchup en ptp a continuacion ***;
; 1  Ejecutar Axis_Rob_Move
; 2  Hacer TouchUp en ptp
; 3  Eliminar Axis_Rob_Move y comentarios

Axis_Rob_Move(1.69,-82.8,66.93,14.32,12.14,193,70,50)

;FOLD PTP pWB90517RS2 Vel=100 % PDAT_MESA Tool[10]:AMF1_G1000 Base[9]:BWB2S2;%{PE}%R 5.5.32,%MKUKATPBASIS,%CMOVE,%VPTP,%P 1:PTP, 2:pWB90517RS2, 3:, 5:100, 7:PDAT_MESA
$BWDSTART=FALSE
PDAT_ACT=PPDAT_MESA
FDAT_ACT=FpWB90517RS2
BAS(#PTP_PARAMS,100)
PTP XpWB90517RS2
;ENDFOLD
;*********************************************************;

;***Axis_Rob_Move de ayuda para aproximarse a dejada ***;
; Borrar tras touchup en LIN de dejada
Axis_Rob_Move(-90.22,-57.13,49.23,-5.44,97.37,193.9,20,50)
;*******************************************************;

PTP_OFFS(XP90517RS2, FP90517RS2, 0, -450, 30, 0, 0, 0, #TOOL, 20, 50, 0.0)

Cicle_Grp_M1000 (Inic_Pla_Right)

;***borrar***;
cyltopos(prg_200)
halt
;************;

LIN_OFFS(XP90517RS2, FP90517RS2, 0, 0, 30, 0, 0, 0, #TOOL, 0.1, 50, 0.0)
LIN_OFFS(XP90517RS2, FP90517RS2, 0, 0, 15, 0, 0, 0, #TOOL, 0.1, 50, 0.0)

Cntr_Grp_M1000 (C05C06,RH)

;FOLD LIN P90517RS2 Vel=0.1 m/s LV020Z0 Tool[10]:AMF1_G1000 Base[9]:BWB2S2;%{PE}%R 5.5.32,%MKUKATPBASIS,%CMOVE,%VLIN,%P 1:LIN, 2:P90517RS2, 3:, 5:0.1, 7:V020Z0
$BWDSTART=FALSE
LDAT_ACT=LV020Z0
FDAT_ACT=FP90517RS2
BAS(#CP_PARAMS,0.1)
LIN XP90517RS2
;ENDFOLD

Cntr_Grp_M1000 (AMF09,RLS)
Cyltopos (PRG_51)
Cntr_Grp_M1000 (C07C08,RH)
Cyltopos (PRG_61)
Cntr_Grp_M1000 (AMF10,RLS)
Cntr_Grp_M1000 (C05C06,FREE)
Cntr_Grp_M1000 (C07C08,FREE)
Cyltopos(PRG_88)
LIN_REL{Z -20}#TOOL
Cyltopos (PRG_105)
LIN_REL{Z -30}#TOOL
Cyltopos (PRG_200)

;*** MOVIMIENTOS DE OFFSETS ***;

LIN_OFFS(XP90517RS2, FP90517RS2, 0, 0, -50, 0, 0, 0, #TOOL, 0.3, 50, 0.0)
LIN_OFFS(XP90517RS2, FP90517RS2, 0, -450, -50, 0, 0, 0, #TOOL, 0.3, 50, 0.0)


;******* MEDICION LASER *******;

LIN_OFFS(XPLAS90517RS2_1, FPLAS90517RS2_1, 0, -200, 0, 0, 0, 0, #TOOL, 0.3, 50, 0.0)

cyltopos (prg_61)

;FOLD LIN PLAS90517RS2_1 Vel=0.3 m/s LV020Z0 Tool[10]:AMF1_G1000 Base[9]:BWB2S2;%{PE}%R 5.5.32,%MKUKATPBASIS,%CMOVE,%VLIN,%P 1:LIN, 2:PLAS90517RS2_1, 3:, 5:0.3, 7:V020Z0
$BWDSTART=FALSE
LDAT_ACT=LV020Z0
FDAT_ACT=FPLAS90517RS2_1
BAS(#CP_PARAMS,0.3)
LIN XPLAS90517RS2_1
;ENDFOLD

;Movimimiento de busqueda con laser
;Search( , )

;FOLD LIN PLAS90517RS2_2 Vel=0.3 m/s LV020Z0 Tool[10]:AMF1_G1000 Base[9]:BWB2S2;%{PE}%R 5.5.32,%MKUKATPBASIS,%CMOVE,%VLIN,%P 1:LIN, 2:PLAS90517RS2_2, 3:, 5:0.3, 7:V020Z0
$BWDSTART=FALSE
LDAT_ACT=LV020Z0
FDAT_ACT=FPLAS90517RS2_2
BAS(#CP_PARAMS,0.3)
LIN XPLAS90517RS2_2
;ENDFOLD


;Movimimiento de busqueda con laser
;Search( , )

LIN_OFFS(XPLAS90517RS2_1, FPLAS90517RS2_1, 0, -200, 0, 0, 0, 0, #TOOL, 0.3, 50, 0.0)

;******************************;

;FOLD PTP pWB90517RS2 Vel=100 % PDAT_MESA Tool[10]:AMF1_G1000 Base[9]:BWB2S2;%{PE}%R 5.5.32,%MKUKATPBASIS,%CMOVE,%VPTP,%P 1:PTP, 2:pWB90517RS2, 3:, 5:100, 7:PDAT_MESA
$BWDSTART=FALSE
PDAT_ACT=PPDAT_MESA
FDAT_ACT=FpWB90517RS2
BAS(#PTP_PARAMS,100)
PTP XpWB90517RS2
;ENDFOLD

;*******************************************************
CASE 90519
;*******************************************************
;*** Utilizar para hacer touchup en ptp a continuacion ***;
; 1  Ejecutar Axis_Rob_Move
; 2  Hacer TouchUp en ptp
; 3  Eliminar Axis_Rob_Move y comentarios

Axis_Rob_Move(1.69,-82.8,66.93,14.32,12.14,193,70,50)

;FOLD PTP pWB90519RS2 Vel=100 % PDAT_MESA Tool[10]:AMF1_G1000 Base[9]:BWB2S2;%{PE}%R 5.5.32,%MKUKATPBASIS,%CMOVE,%VPTP,%P 1:PTP, 2:pWB90519RS2, 3:, 5:100, 7:PDAT_MESA
$BWDSTART=FALSE
PDAT_ACT=PPDAT_MESA
FDAT_ACT=FpWB90519RS2
BAS(#PTP_PARAMS,100)
PTP XpWB90519RS2
;ENDFOLD
;*********************************************************;

;***Axis_Rob_Move de ayuda para aproximarse a dejada ***;
; Borrar tras touchup en LIN de dejada
Axis_Rob_Move(-90.22,-57.13,49.23,-5.44,97.37,193.9,20,50)
;*******************************************************;

PTP_OFFS(XP90519RS2, FP90519RS2, 0, -450, 30, 0, 0, 0, #TOOL, 20, 50, 0.0)

Cicle_Grp_M1000 (Inic_Pla_Right)

;***borrar***;
cyltopos(prg_200)
halt
;************;

LIN_OFFS(XP90519RS2, FP90519RS2, 0, 0, 30, 0, 0, 0, #TOOL, 0.1, 50, 0.0)
LIN_OFFS(XP90519RS2, FP90519RS2, 0, 0, 15, 0, 0, 0, #TOOL, 0.1, 50, 0.0)

Cntr_Grp_M1000 (C05C06,RH)

;FOLD LIN P90519RS2 Vel=0.1 m/s LV020Z0 Tool[10]:AMF1_G1000 Base[9]:BWB2S2;%{PE}%R 5.5.32,%MKUKATPBASIS,%CMOVE,%VLIN,%P 1:LIN, 2:P90519RS2, 3:, 5:0.1, 7:V020Z0
$BWDSTART=FALSE
LDAT_ACT=LV020Z0
FDAT_ACT=FP90519RS2
BAS(#CP_PARAMS,0.1)
LIN XP90519RS2
;ENDFOLD

Cntr_Grp_M1000 (AMF09,RLS)
Cyltopos (PRG_51)
Cntr_Grp_M1000 (C07C08,RH)
Cyltopos (PRG_61)
Cntr_Grp_M1000 (AMF10,RLS)
Cntr_Grp_M1000 (C05C06,FREE)
Cntr_Grp_M1000 (C07C08,FREE)
Cyltopos(PRG_88)
LIN_REL{Z -20}#TOOL
Cyltopos (PRG_105)
LIN_REL{Z -30}#TOOL
Cyltopos (PRG_200)

;*** MOVIMIENTOS DE OFFSETS ***;

LIN_OFFS(XP90519RS2, FP90519RS2, 0, 0, -50, 0, 0, 0, #TOOL, 0.3, 50, 0.0)
LIN_OFFS(XP90519RS2, FP90519RS2, 0, -450, -50, 0, 0, 0, #TOOL, 0.3, 50, 0.0)


;******* MEDICION LASER *******;

LIN_OFFS(XPLAS90519RS2_1, FPLAS90519RS2_1, 0, -200, 0, 0, 0, 0, #TOOL, 0.3, 50, 0.0)

cyltopos (prg_61)

;FOLD LIN PLAS90519RS2_1 Vel=0.3 m/s LV020Z0 Tool[10]:AMF1_G1000 Base[9]:BWB2S2;%{PE}%R 5.5.32,%MKUKATPBASIS,%CMOVE,%VLIN,%P 1:LIN, 2:PLAS90519RS2_1, 3:, 5:0.3, 7:V020Z0
$BWDSTART=FALSE
LDAT_ACT=LV020Z0
FDAT_ACT=FPLAS90519RS2_1
BAS(#CP_PARAMS,0.3)
LIN XPLAS90519RS2_1
;ENDFOLD

;Movimimiento de busqueda con laser
;Search( , )

;FOLD LIN PLAS90519RS2_2 Vel=0.3 m/s LV020Z0 Tool[10]:AMF1_G1000 Base[9]:BWB2S2;%{PE}%R 5.5.32,%MKUKATPBASIS,%CMOVE,%VLIN,%P 1:LIN, 2:PLAS90519RS2_2, 3:, 5:0.3, 7:V020Z0
$BWDSTART=FALSE
LDAT_ACT=LV020Z0
FDAT_ACT=FPLAS90519RS2_2
BAS(#CP_PARAMS,0.3)
LIN XPLAS90519RS2_2
;ENDFOLD


;Movimimiento de busqueda con laser
;Search( , )

LIN_OFFS(XPLAS90519RS2_1, FPLAS90519RS2_1, 0, -200, 0, 0, 0, 0, #TOOL, 0.3, 50, 0.0)

;******************************;

;FOLD PTP pWB90519RS2 Vel=100 % PDAT_MESA Tool[10]:AMF1_G1000 Base[9]:BWB2S2;%{PE}%R 5.5.32,%MKUKATPBASIS,%CMOVE,%VPTP,%P 1:PTP, 2:pWB90519RS2, 3:, 5:100, 7:PDAT_MESA
$BWDSTART=FALSE
PDAT_ACT=PPDAT_MESA
FDAT_ACT=FpWB90519RS2
BAS(#PTP_PARAMS,100)
PTP XpWB90519RS2
;ENDFOLD

;*******************************************************
CASE 90521
;*******************************************************
;*** Utilizar para hacer touchup en ptp a continuacion ***;
; 1  Ejecutar Axis_Rob_Move
; 2  Hacer TouchUp en ptp
; 3  Eliminar Axis_Rob_Move y comentarios

Axis_Rob_Move(1.69,-82.8,66.93,14.32,12.14,193,70,50)

;FOLD PTP pWB90521RS2 Vel=100 % PDAT_MESA Tool[10]:AMF1_G1000 Base[9]:BWB2S2;%{PE}%R 5.5.32,%MKUKATPBASIS,%CMOVE,%VPTP,%P 1:PTP, 2:pWB90521RS2, 3:, 5:100, 7:PDAT_MESA
$BWDSTART=FALSE
PDAT_ACT=PPDAT_MESA
FDAT_ACT=FpWB90521RS2
BAS(#PTP_PARAMS,100)
PTP XpWB90521RS2
;ENDFOLD
;*********************************************************;

;***Axis_Rob_Move de ayuda para aproximarse a dejada ***;
; Borrar tras touchup en LIN de dejada
Axis_Rob_Move(-90.22,-57.13,49.23,-5.44,97.37,193.9,20,50)
;*******************************************************;

PTP_OFFS(XP90521RS2, FP90521RS2, 0, -450, 30, 0, 0, 0, #TOOL, 20, 50, 0.0)

Cicle_Grp_M1000 (Inic_Pla_Right)

;***borrar***;
cyltopos(prg_200)
halt
;************;

LIN_OFFS(XP90521RS2, FP90521RS2, 0, 0, 30, 0, 0, 0, #TOOL, 0.1, 50, 0.0)
LIN_OFFS(XP90521RS2, FP90521RS2, 0, 0, 15, 0, 0, 0, #TOOL, 0.1, 50, 0.0)

Cntr_Grp_M1000 (C05C06,RH)

;FOLD LIN P90521RS2 Vel=0.1 m/s LV020Z0 Tool[10]:AMF1_G1000 Base[9]:BWB2S2;%{PE}%R 5.5.32,%MKUKATPBASIS,%CMOVE,%VLIN,%P 1:LIN, 2:P90521RS2, 3:, 5:0.1, 7:V020Z0
$BWDSTART=FALSE
LDAT_ACT=LV020Z0
FDAT_ACT=FP90521RS2
BAS(#CP_PARAMS,0.1)
LIN XP90521RS2
;ENDFOLD

Cntr_Grp_M1000 (AMF09,RLS)
Cyltopos (PRG_51)
Cntr_Grp_M1000 (C07C08,RH)
Cyltopos (PRG_61)
Cntr_Grp_M1000 (AMF10,RLS)
Cntr_Grp_M1000 (C05C06,FREE)
Cntr_Grp_M1000 (C07C08,FREE)
Cyltopos(PRG_88)
LIN_REL{Z -20}#TOOL
Cyltopos (PRG_105)
LIN_REL{Z -30}#TOOL
Cyltopos (PRG_200)

;*** MOVIMIENTOS DE OFFSETS ***;

LIN_OFFS(XP90521RS2, FP90521RS2, 0, 0, -50, 0, 0, 0, #TOOL, 0.3, 50, 0.0)
LIN_OFFS(XP90521RS2, FP90521RS2, 0, -450, -50, 0, 0, 0, #TOOL, 0.3, 50, 0.0)


;******* MEDICION LASER *******;

LIN_OFFS(XPLAS90521RS2_1, FPLAS90521RS2_1, 0, -200, 0, 0, 0, 0, #TOOL, 0.3, 50, 0.0)

cyltopos (prg_61)

;FOLD LIN PLAS90521RS2_1 Vel=0.3 m/s LV020Z0 Tool[10]:AMF1_G1000 Base[9]:BWB2S2;%{PE}%R 5.5.32,%MKUKATPBASIS,%CMOVE,%VLIN,%P 1:LIN, 2:PLAS90521RS2_1, 3:, 5:0.3, 7:V020Z0
$BWDSTART=FALSE
LDAT_ACT=LV020Z0
FDAT_ACT=FPLAS90521RS2_1
BAS(#CP_PARAMS,0.3)
LIN XPLAS90521RS2_1
;ENDFOLD

;Movimimiento de busqueda con laser
;Search( , )

;FOLD LIN PLAS90521RS2_2 Vel=0.3 m/s LV020Z0 Tool[10]:AMF1_G1000 Base[9]:BWB2S2;%{PE}%R 5.5.32,%MKUKATPBASIS,%CMOVE,%VLIN,%P 1:LIN, 2:PLAS90521RS2_2, 3:, 5:0.3, 7:V020Z0
$BWDSTART=FALSE
LDAT_ACT=LV020Z0
FDAT_ACT=FPLAS90521RS2_2
BAS(#CP_PARAMS,0.3)
LIN XPLAS90521RS2_2
;ENDFOLD


;Movimimiento de busqueda con laser
;Search( , )

LIN_OFFS(XPLAS90521RS2_1, FPLAS90521RS2_1, 0, -200, 0, 0, 0, 0, #TOOL, 0.3, 50, 0.0)

;******************************;

;FOLD PTP pWB90521RS2 Vel=100 % PDAT_MESA Tool[10]:AMF1_G1000 Base[9]:BWB2S2;%{PE}%R 5.5.32,%MKUKATPBASIS,%CMOVE,%VPTP,%P 1:PTP, 2:pWB90521RS2, 3:, 5:100, 7:PDAT_MESA
$BWDSTART=FALSE
PDAT_ACT=PPDAT_MESA
FDAT_ACT=FpWB90521RS2
BAS(#PTP_PARAMS,100)
PTP XpWB90521RS2
;ENDFOLD

;*******************************************************
CASE 90523
;*******************************************************
;*** Utilizar para hacer touchup en ptp a continuacion ***;
; 1  Ejecutar Axis_Rob_Move
; 2  Hacer TouchUp en ptp
; 3  Eliminar Axis_Rob_Move y comentarios

Axis_Rob_Move(1.69,-82.8,66.93,14.32,12.14,193,70,50)

;FOLD PTP pWB90523RS2 Vel=100 % PDAT_MESA Tool[10]:AMF1_G1000 Base[9]:BWB2S2;%{PE}%R 5.5.32,%MKUKATPBASIS,%CMOVE,%VPTP,%P 1:PTP, 2:pWB90523RS2, 3:, 5:100, 7:PDAT_MESA
$BWDSTART=FALSE
PDAT_ACT=PPDAT_MESA
FDAT_ACT=FpWB90523RS2
BAS(#PTP_PARAMS,100)
PTP XpWB90523RS2
;ENDFOLD
;*********************************************************;

;***Axis_Rob_Move de ayuda para aproximarse a dejada ***;
; Borrar tras touchup en LIN de dejada
Axis_Rob_Move(-90.22,-57.13,49.23,-5.44,97.37,193.9,20,50)
;*******************************************************;

PTP_OFFS(XP90523RS2, FP90523RS2, 0, -450, 30, 0, 0, 0, #TOOL, 20, 50, 0.0)

Cicle_Grp_M1000 (Inic_Pla_Right)

;***borrar***;
cyltopos(prg_200)
halt
;************;

LIN_OFFS(XP90523RS2, FP90523RS2, 0, 0, 30, 0, 0, 0, #TOOL, 0.1, 50, 0.0)
LIN_OFFS(XP90523RS2, FP90523RS2, 0, 0, 15, 0, 0, 0, #TOOL, 0.1, 50, 0.0)

Cntr_Grp_M1000 (C05C06,RH)

;FOLD LIN P90523RS2 Vel=0.1 m/s LV020Z0 Tool[10]:AMF1_G1000 Base[9]:BWB2S2;%{PE}%R 5.5.32,%MKUKATPBASIS,%CMOVE,%VLIN,%P 1:LIN, 2:P90523RS2, 3:, 5:0.1, 7:V020Z0
$BWDSTART=FALSE
LDAT_ACT=LV020Z0
FDAT_ACT=FP90523RS2
BAS(#CP_PARAMS,0.1)
LIN XP90523RS2
;ENDFOLD

Cntr_Grp_M1000 (AMF09,RLS)
Cyltopos (PRG_51)
Cntr_Grp_M1000 (C07C08,RH)
Cyltopos (PRG_61)
Cntr_Grp_M1000 (AMF10,RLS)
Cntr_Grp_M1000 (C05C06,FREE)
Cntr_Grp_M1000 (C07C08,FREE)
Cyltopos(PRG_88)
LIN_REL{Z -20}#TOOL
Cyltopos (PRG_105)
LIN_REL{Z -30}#TOOL
Cyltopos (PRG_200)

;*** MOVIMIENTOS DE OFFSETS ***;

LIN_OFFS(XP90523RS2, FP90523RS2, 0, 0, -50, 0, 0, 0, #TOOL, 0.3, 50, 0.0)
LIN_OFFS(XP90523RS2, FP90523RS2, 0, -450, -50, 0, 0, 0, #TOOL, 0.3, 50, 0.0)


;******* MEDICION LASER *******;

LIN_OFFS(XPLAS90523RS2_1, FPLAS90523RS2_1, 0, -200, 0, 0, 0, 0, #TOOL, 0.3, 50, 0.0)

cyltopos (prg_61)

;FOLD LIN PLAS90523RS2_1 Vel=0.3 m/s LV020Z0 Tool[10]:AMF1_G1000 Base[9]:BWB2S2;%{PE}%R 5.5.32,%MKUKATPBASIS,%CMOVE,%VLIN,%P 1:LIN, 2:PLAS90523RS2_1, 3:, 5:0.3, 7:V020Z0
$BWDSTART=FALSE
LDAT_ACT=LV020Z0
FDAT_ACT=FPLAS90523RS2_1
BAS(#CP_PARAMS,0.3)
LIN XPLAS90523RS2_1
;ENDFOLD

;Movimimiento de busqueda con laser
;Search( , )

;FOLD LIN PLAS90523RS2_2 Vel=0.3 m/s LV020Z0 Tool[10]:AMF1_G1000 Base[9]:BWB2S2;%{PE}%R 5.5.32,%MKUKATPBASIS,%CMOVE,%VLIN,%P 1:LIN, 2:PLAS90523RS2_2, 3:, 5:0.3, 7:V020Z0
$BWDSTART=FALSE
LDAT_ACT=LV020Z0
FDAT_ACT=FPLAS90523RS2_2
BAS(#CP_PARAMS,0.3)
LIN XPLAS90523RS2_2
;ENDFOLD


;Movimimiento de busqueda con laser
;Search( , )

LIN_OFFS(XPLAS90523RS2_1, FPLAS90523RS2_1, 0, -200, 0, 0, 0, 0, #TOOL, 0.3, 50, 0.0)

;******************************;

;FOLD PTP pWB90523RS2 Vel=100 % PDAT_MESA Tool[10]:AMF1_G1000 Base[9]:BWB2S2;%{PE}%R 5.5.32,%MKUKATPBASIS,%CMOVE,%VPTP,%P 1:PTP, 2:pWB90523RS2, 3:, 5:100, 7:PDAT_MESA
$BWDSTART=FALSE
PDAT_ACT=PPDAT_MESA
FDAT_ACT=FpWB90523RS2
BAS(#PTP_PARAMS,100)
PTP XpWB90523RS2
;ENDFOLD

ENDSWITCH
END

--- nplacestr5RS2.dat ---
DEFDAT nplacestr5RS2
;FOLD EXTERNAL DECLARATIONS;%{PE}%MKUKATPBASIS,%CEXT,%VCOMMON,%P
;FOLD BASISTECH EXT;%{PE}%MKUKATPBASIS,%CEXT,%VEXT,%P
EXT  BAS (BAS_COMMAND  :IN,REAL  :IN )
DECL INT SUCCESS
;ENDFOLD (BASISTECH EXT)
;FOLD USER EXT;%{E}%MKUKATPUSER,%CEXT,%VEXT,%P
;Make here your modifications

;ENDFOLD (USER EXT)
;ENDFOLD (EXTERNAL DECLARATIONS)
DECL E6POS XpWB90501RS2={X 0,Y 0,Z 0,A 0,B 0,C 0,S 2,T 10,E1 0.0,E2 0.0,E3 0.0,E4 0.0,E5 0.0,E6 0.0}
DECL FDAT FpWB90501RS2={TOOL_NO 10,BASE_NO 9,IPO_FRAME #BASE,POINT2[] " ",TQ_STATE FALSE}
;
DECL E6POS XP90501RS2={X 0,Y 0,Z 0,A 0,B 0,C 0,S 2,T 10,E1 0.0,E2 0.0,E3 0.0,E4 0.0,E5 0.0,E6 0.0}
DECL FDAT FP90501RS2={TOOL_NO 10,BASE_NO 9,IPO_FRAME #BASE,POINT2[] " ",TQ_STATE FALSE}
;
DECL E6POS XPLAS90501RS2_1={X 0,Y 0,Z 0,A 0,B 0,C 0,S 2,T 10,E1 0.0,E2 0.0,E3 0.0,E4 0.0,E5 0.0,E6 0.0}
DECL FDAT FPLAS90501RS2_1={TOOL_NO 10,BASE_NO 9,IPO_FRAME #BASE,POINT2[] " ",TQ_STATE FALSE}
DECL E6POS XPLAS90501RS2_2={X 0,Y 0,Z 0,A 0,B 0,C 0,S 2,T 10,E1 0.0,E2 0.0,E3 0.0,E4 0.0,E5 0.0,E6 0.0}
DECL FDAT FPLAS90501RS2_2={TOOL_NO 10,BASE_NO 9,IPO_FRAME #BASE,POINT2[] " ",TQ_STATE FALSE}
;
DECL E6POS XpWB90503RS2={X 0,Y 0,Z 0,A 0,B 0,C 0,S 2,T 10,E1 0.0,E2 0.0,E3 0.0,E4 0.0,E5 0.0,E6 0.0}
DECL FDAT FpWB90503RS2={TOOL_NO 10,BASE_NO 9,IPO_FRAME #BASE,POINT2[] " ",TQ_STATE FALSE}
;
DECL E6POS XP90503RS2={X 0,Y 0,Z 0,A 0,B 0,C 0,S 2,T 10,E1 0.0,E2 0.0,E3 0.0,E4 0.0,E5 0.0,E6 0.0}
DECL FDAT FP90503RS2={TOOL_NO 10,BASE_NO 9,IPO_FRAME #BASE,POINT2[] " ",TQ_STATE FALSE}
;
DECL E6POS XPLAS90503RS2_1={X 0,Y 0,Z 0,A 0,B 0,C 0,S 2,T 10,E1 0.0,E2 0.0,E3 0.0,E4 0.0,E5 0.0,E6 0.0}
DECL FDAT FPLAS90503RS2_1={TOOL_NO 10,BASE_NO 9,IPO_FRAME #BASE,POINT2[] " ",TQ_STATE FALSE}
DECL E6POS XPLAS90503RS2_2={X 0,Y 0,Z 0,A 0,B 0,C 0,S 2,T 10,E1 0.0,E2 0.0,E3 0.0,E4 0.0,E5 0.0,E6 0.0}
DECL FDAT FPLAS90503RS2_2={TOOL_NO 10,BASE_NO 9,IPO_FRAME #BASE,POINT2[] " ",TQ_STATE FALSE}
;
DECL E6POS XpWB90505RS2={X 0,Y 0,Z 0,A 0,B 0,C 0,S 2,T 10,E1 0.0,E2 0.0,E3 0.0,E4 0.0,E5 0.0,E6 0.0}
DECL FDAT FpWB90505RS2={TOOL_NO 10,BASE_NO 9,IPO_FRAME #BASE,POINT2[] " ",TQ_STATE FALSE}
;
DECL E6POS XP90505RS2={X 0,Y 0,Z 0,A 0,B 0,C 0,S 2,T 10,E1 0.0,E2 0.0,E3 0.0,E4 0.0,E5 0.0,E6 0.0}
DECL FDAT FP90505RS2={TOOL_NO 10,BASE_NO 9,IPO_FRAME #BASE,POINT2[] " ",TQ_STATE FALSE}
;
DECL E6POS XPLAS90505RS2_1={X 0,Y 0,Z 0,A 0,B 0,C 0,S 2,T 10,E1 0.0,E2 0.0,E3 0.0,E4 0.0,E5 0.0,E6 0.0}
DECL FDAT FPLAS90505RS2_1={TOOL_NO 10,BASE_NO 9,IPO_FRAME #BASE,POINT2[] " ",TQ_STATE FALSE}
DECL E6POS XPLAS90505RS2_2={X 0,Y 0,Z 0,A 0,B 0,C 0,S 2,T 10,E1 0.0,E2 0.0,E3 0.0,E4 0.0,E5 0.0,E6 0.0}
DECL FDAT FPLAS90505RS2_2={TOOL_NO 10,BASE_NO 9,IPO_FRAME #BASE,POINT2[] " ",TQ_STATE FALSE}
;
DECL E6POS XpWB90507RS2={X 0,Y 0,Z 0,A 0,B 0,C 0,S 2,T 10,E1 0.0,E2 0.0,E3 0.0,E4 0.0,E5 0.0,E6 0.0}
DECL FDAT FpWB90507RS2={TOOL_NO 10,BASE_NO 9,IPO_FRAME #BASE,POINT2[] " ",TQ_STATE FALSE}
;
DECL E6POS XP90507RS2={X 0,Y 0,Z 0,A 0,B 0,C 0,S 2,T 10,E1 0.0,E2 0.0,E3 0.0,E4 0.0,E5 0.0,E6 0.0}
DECL FDAT FP90507RS2={TOOL_NO 10,BASE_NO 9,IPO_FRAME #BASE,POINT2[] " ",TQ_STATE FALSE}
;
DECL E6POS XPLAS90507RS2_1={X 0,Y 0,Z 0,A 0,B 0,C 0,S 2,T 10,E1 0.0,E2 0.0,E3 0.0,E4 0.0,E5 0.0,E6 0.0}
DECL FDAT FPLAS90507RS2_1={TOOL_NO 10,BASE_NO 9,IPO_FRAME #BASE,POINT2[] " ",TQ_STATE FALSE}
DECL E6POS XPLAS90507RS2_2={X 0,Y 0,Z 0,A 0,B 0,C 0,S 2,T 10,E1 0.0,E2 0.0,E3 0.0,E4 0.0,E5 0.0,E6 0.0}
DECL FDAT FPLAS90507RS2_2={TOOL_NO 10,BASE_NO 9,IPO_FRAME #BASE,POINT2[] " ",TQ_STATE FALSE}
;
DECL E6POS XpWB90509RS2={X 0,Y 0,Z 0,A 0,B 0,C 0,S 2,T 10,E1 0.0,E2 0.0,E3 0.0,E4 0.0,E5 0.0,E6 0.0}
DECL FDAT FpWB90509RS2={TOOL_NO 10,BASE_NO 9,IPO_FRAME #BASE,POINT2[] " ",TQ_STATE FALSE}
;
DECL E6POS XP90509RS2={X 0,Y 0,Z 0,A 0,B 0,C 0,S 2,T 10,E1 0.0,E2 0.0,E3 0.0,E4 0.0,E5 0.0,E6 0.0}
DECL FDAT FP90509RS2={TOOL_NO 10,BASE_NO 9,IPO_FRAME #BASE,POINT2[] " ",TQ_STATE FALSE}
;
DECL E6POS XPLAS90509RS2_1={X 0,Y 0,Z 0,A 0,B 0,C 0,S 2,T 10,E1 0.0,E2 0.0,E3 0.0,E4 0.0,E5 0.0,E6 0.0}
DECL FDAT FPLAS90509RS2_1={TOOL_NO 10,BASE_NO 9,IPO_FRAME #BASE,POINT2[] " ",TQ_STATE FALSE}
DECL E6POS XPLAS90509RS2_2={X 0,Y 0,Z 0,A 0,B 0,C 0,S 2,T 10,E1 0.0,E2 0.0,E3 0.0,E4 0.0,E5 0.0,E6 0.0}
DECL FDAT FPLAS90509RS2_2={TOOL_NO 10,BASE_NO 9,IPO_FRAME #BASE,POINT2[] " ",TQ_STATE FALSE}
;
DECL E6POS XpWB90511RS2={X 0,Y 0,Z 0,A 0,B 0,C 0,S 2,T 10,E1 0.0,E2 0.0,E3 0.0,E4 0.0,E5 0.0,E6 0.0}
DECL FDAT FpWB90511RS2={TOOL_NO 10,BASE_NO 9,IPO_FRAME #BASE,POINT2[] " ",TQ_STATE FALSE}
;
DECL E6POS XP90511RS2={X 0,Y 0,Z 0,A 0,B 0,C 0,S 2,T 10,E1 0.0,E2 0.0,E3 0.0,E4 0.0,E5 0.0,E6 0.0}
DECL FDAT FP90511RS2={TOOL_NO 10,BASE_NO 9,IPO_FRAME #BASE,POINT2[] " ",TQ_STATE FALSE}
;
DECL E6POS XPLAS90511RS2_1={X 0,Y 0,Z 0,A 0,B 0,C 0,S 2,T 10,E1 0.0,E2 0.0,E3 0.0,E4 0.0,E5 0.0,E6 0.0}
DECL FDAT FPLAS90511RS2_1={TOOL_NO 10,BASE_NO 9,IPO_FRAME #BASE,POINT2[] " ",TQ_STATE FALSE}
DECL E6POS XPLAS90511RS2_2={X 0,Y 0,Z 0,A 0,B 0,C 0,S 2,T 10,E1 0.0,E2 0.0,E3 0.0,E4 0.0,E5 0.0,E6 0.0}
DECL FDAT FPLAS90511RS2_2={TOOL_NO 10,BASE_NO 9,IPO_FRAME #BASE,POINT2[] " ",TQ_STATE FALSE}
;
DECL E6POS XpWB90513RS2={X 0,Y 0,Z 0,A 0,B 0,C 0,S 2,T 10,E1 0.0,E2 0.0,E3 0.0,E4 0.0,E5 0.0,E6 0.0}
DECL FDAT FpWB90513RS2={TOOL_NO 10,BASE_NO 9,IPO_FRAME #BASE,POINT2[] " ",TQ_STATE FALSE}
;
DECL E6POS XP90513RS2={X 0,Y 0,Z 0,A 0,B 0,C 0,S 2,T 10,E1 0.0,E2 0.0,E3 0.0,E4 0.0,E5 0.0,E6 0.0}
DECL FDAT FP90513RS2={TOOL_NO 10,BASE_NO 9,IPO_FRAME #BASE,POINT2[] " ",TQ_STATE FALSE}
;
DECL E6POS XPLAS90513RS2_1={X 0,Y 0,Z 0,A 0,B 0,C 0,S 2,T 10,E1 0.0,E2 0.0,E3 0.0,E4 0.0,E5 0.0,E6 0.0}
DECL FDAT FPLAS90513RS2_1={TOOL_NO 10,BASE_NO 9,IPO_FRAME #BASE,POINT2[] " ",TQ_STATE FALSE}
DECL E6POS XPLAS90513RS2_2={X 0,Y 0,Z 0,A 0,B 0,C 0,S 2,T 10,E1 0.0,E2 0.0,E3 0.0,E4 0.0,E5 0.0,E6 0.0}
DECL FDAT FPLAS90513RS2_2={TOOL_NO 10,BASE_NO 9,IPO_FRAME #BASE,POINT2[] " ",TQ_STATE FALSE}
;
DECL E6POS XpWB90515RS2={X 0,Y 0,Z 0,A 0,B 0,C 0,S 2,T 10,E1 0.0,E2 0.0,E3 0.0,E4 0.0,E5 0.0,E6 0.0}
DECL FDAT FpWB90515RS2={TOOL_NO 10,BASE_NO 9,IPO_FRAME #BASE,POINT2[] " ",TQ_STATE FALSE}
;
DECL E6POS XP90515RS2={X 0,Y 0,Z 0,A 0,B 0,C 0,S 2,T 10,E1 0.0,E2 0.0,E3 0.0,E4 0.0,E5 0.0,E6 0.0}
DECL FDAT FP90515RS2={TOOL_NO 10,BASE_NO 9,IPO_FRAME #BASE,POINT2[] " ",TQ_STATE FALSE}
;
DECL E6POS XPLAS90515RS2_1={X 0,Y 0,Z 0,A 0,B 0,C 0,S 2,T 10,E1 0.0,E2 0.0,E3 0.0,E4 0.0,E5 0.0,E6 0.0}
DECL FDAT FPLAS90515RS2_1={TOOL_NO 10,BASE_NO 9,IPO_FRAME #BASE,POINT2[] " ",TQ_STATE FALSE}
DECL E6POS XPLAS90515RS2_2={X 0,Y 0,Z 0,A 0,B 0,C 0,S 2,T 10,E1 0.0,E2 0.0,E3 0.0,E4 0.0,E5 0.0,E6 0.0}
DECL FDAT FPLAS90515RS2_2={TOOL_NO 10,BASE_NO 9,IPO_FRAME #BASE,POINT2[] " ",TQ_STATE FALSE}
;
DECL E6POS XpWB90517RS2={X 0,Y 0,Z 0,A 0,B 0,C 0,S 2,T 10,E1 0.0,E2 0.0,E3 0.0,E4 0.0,E5 0.0,E6 0.0}
DECL FDAT FpWB90517RS2={TOOL_NO 10,BASE_NO 9,IPO_FRAME #BASE,POINT2[] " ",TQ_STATE FALSE}
;
DECL E6POS XP90517RS2={X 0,Y 0,Z 0,A 0,B 0,C 0,S 2,T 10,E1 0.0,E2 0.0,E3 0.0,E4 0.0,E5 0.0,E6 0.0}
DECL FDAT FP90517RS2={TOOL_NO 10,BASE_NO 9,IPO_FRAME #BASE,POINT2[] " ",TQ_STATE FALSE}
;
DECL E6POS XPLAS90517RS2_1={X 0,Y 0,Z 0,A 0,B 0,C 0,S 2,T 10,E1 0.0,E2 0.0,E3 0.0,E4 0.0,E5 0.0,E6 0.0}
DECL FDAT FPLAS90517RS2_1={TOOL_NO 10,BASE_NO 9,IPO_FRAME #BASE,POINT2[] " ",TQ_STATE FALSE}
DECL E6POS XPLAS90517RS2_2={X 0,Y 0,Z 0,A 0,B 0,C 0,S 2,T 10,E1 0.0,E2 0.0,E3 0.0,E4 0.0,E5 0.0,E6 0.0}
DECL FDAT FPLAS90517RS2_2={TOOL_NO 10,BASE_NO 9,IPO_FRAME #BASE,POINT2[] " ",TQ_STATE FALSE}
;
DECL E6POS XpWB90519RS2={X 0,Y 0,Z 0,A 0,B 0,C 0,S 2,T 10,E1 0.0,E2 0.0,E3 0.0,E4 0.0,E5 0.0,E6 0.0}
DECL FDAT FpWB90519RS2={TOOL_NO 10,BASE_NO 9,IPO_FRAME #BASE,POINT2[] " ",TQ_STATE FALSE}
;
DECL E6POS XP90519RS2={X 0,Y 0,Z 0,A 0,B 0,C 0,S 2,T 10,E1 0.0,E2 0.0,E3 0.0,E4 0.0,E5 0.0,E6 0.0}
DECL FDAT FP90519RS2={TOOL_NO 10,BASE_NO 9,IPO_FRAME #BASE,POINT2[] " ",TQ_STATE FALSE}
;
DECL E6POS XPLAS90519RS2_1={X 0,Y 0,Z 0,A 0,B 0,C 0,S 2,T 10,E1 0.0,E2 0.0,E3 0.0,E4 0.0,E5 0.0,E6 0.0}
DECL FDAT FPLAS90519RS2_1={TOOL_NO 10,BASE_NO 9,IPO_FRAME #BASE,POINT2[] " ",TQ_STATE FALSE}
DECL E6POS XPLAS90519RS2_2={X 0,Y 0,Z 0,A 0,B 0,C 0,S 2,T 10,E1 0.0,E2 0.0,E3 0.0,E4 0.0,E5 0.0,E6 0.0}
DECL FDAT FPLAS90519RS2_2={TOOL_NO 10,BASE_NO 9,IPO_FRAME #BASE,POINT2[] " ",TQ_STATE FALSE}
;
DECL E6POS XpWB90521RS2={X 0,Y 0,Z 0,A 0,B 0,C 0,S 2,T 10,E1 0.0,E2 0.0,E3 0.0,E4 0.0,E5 0.0,E6 0.0}
DECL FDAT FpWB90521RS2={TOOL_NO 10,BASE_NO 9,IPO_FRAME #BASE,POINT2[] " ",TQ_STATE FALSE}
;
DECL E6POS XP90521RS2={X 0,Y 0,Z 0,A 0,B 0,C 0,S 2,T 10,E1 0.0,E2 0.0,E3 0.0,E4 0.0,E5 0.0,E6 0.0}
DECL FDAT FP90521RS2={TOOL_NO 10,BASE_NO 9,IPO_FRAME #BASE,POINT2[] " ",TQ_STATE FALSE}
;
DECL E6POS XPLAS90521RS2_1={X 0,Y 0,Z 0,A 0,B 0,C 0,S 2,T 10,E1 0.0,E2 0.0,E3 0.0,E4 0.0,E5 0.0,E6 0.0}
DECL FDAT FPLAS90521RS2_1={TOOL_NO 10,BASE_NO 9,IPO_FRAME #BASE,POINT2[] " ",TQ_STATE FALSE}
DECL E6POS XPLAS90521RS2_2={X 0,Y 0,Z 0,A 0,B 0,C 0,S 2,T 10,E1 0.0,E2 0.0,E3 0.0,E4 0.0,E5 0.0,E6 0.0}
DECL FDAT FPLAS90521RS2_2={TOOL_NO 10,BASE_NO 9,IPO_FRAME #BASE,POINT2[] " ",TQ_STATE FALSE}
;
DECL E6POS XpWB90523RS2={X 0,Y 0,Z 0,A 0,B 0,C 0,S 2,T 10,E1 0.0,E2 0.0,E3 0.0,E4 0.0,E5 0.0,E6 0.0}
DECL FDAT FpWB90523RS2={TOOL_NO 10,BASE_NO 9,IPO_FRAME #BASE,POINT2[] " ",TQ_STATE FALSE}
;
DECL E6POS XP90523RS2={X 0,Y 0,Z 0,A 0,B 0,C 0,S 2,T 10,E1 0.0,E2 0.0,E3 0.0,E4 0.0,E5 0.0,E6 0.0}
DECL FDAT FP90523RS2={TOOL_NO 10,BASE_NO 9,IPO_FRAME #BASE,POINT2[] " ",TQ_STATE FALSE}
;
DECL E6POS XPLAS90523RS2_1={X 0,Y 0,Z 0,A 0,B 0,C 0,S 2,T 10,E1 0.0,E2 0.0,E3 0.0,E4 0.0,E5 0.0,E6 0.0}
DECL FDAT FPLAS90523RS2_1={TOOL_NO 10,BASE_NO 9,IPO_FRAME #BASE,POINT2[] " ",TQ_STATE FALSE}
DECL E6POS XPLAS90523RS2_2={X 0,Y 0,Z 0,A 0,B 0,C 0,S 2,T 10,E1 0.0,E2 0.0,E3 0.0,E4 0.0,E5 0.0,E6 0.0}
DECL FDAT FPLAS90523RS2_2={TOOL_NO 10,BASE_NO 9,IPO_FRAME #BASE,POINT2[] " ",TQ_STATE FALSE}
;
ENDDAT
